TYPE ST_ViciStatus :
STRUCT
	sViciReq			: STRING;
	sViciReply		:STRING;
	iCurrPos				: INT;
	iReqPos		:	INT;
	xPosValid	:	BOOL;
	(*iAddress				:INT;*)
	(* Do not use this address. If you do, the driver
	will overwrite this address with zero each time
	it runs, as the status is an input, not in_out *)			
END_STRUCT
END_TYPE

(* stored: Version 1.1.0.1, ProductVersion 3.1.0.24
   DUT ST_ViciStatus: Id {3cbe973d-3413-4383-8a07-6d21d8bf92fd} *)
